INTERFACE ITF_EM_Turning

END_INTERFACE

(* stored: Version 1.1.0.1, ProductVersion 3.1.4024.12
   Itf ITF_EM_Turning: Id {f325c623-acde-4b57-ba7d-be34b8f9dfd4} *)
